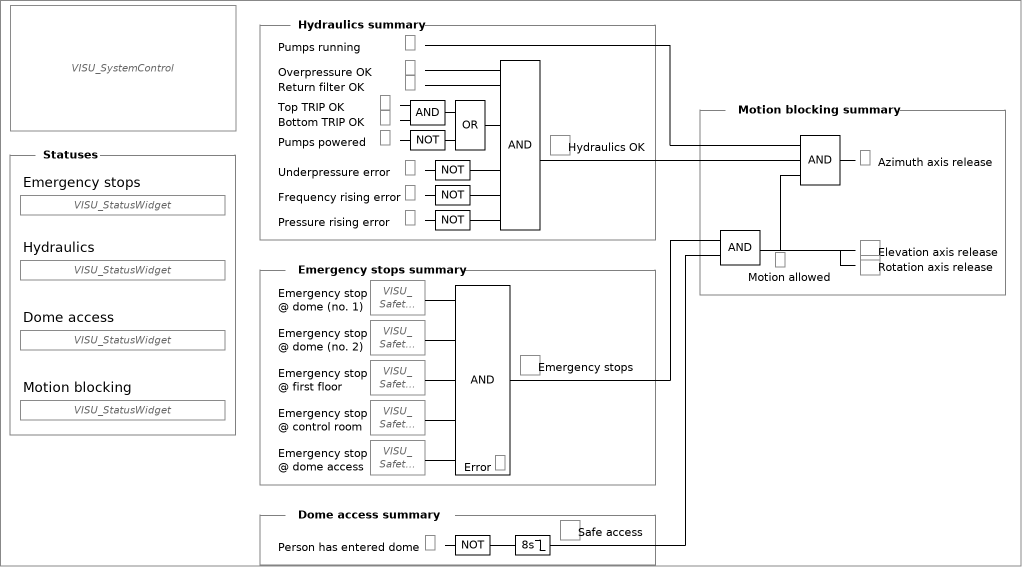
VISUALIZATION VISU_SafetyOverview  // 1022x567
VAR_IN_OUT
	ref : Safety;
    widget : SafetyWidget;
END_VAR
    Polyline (900,110) (1005,110) (1005,295) (700,295) (700,110) (725,110)
    Polyline (455,515) (655,515) (655,565) (260,565) (260,515) (285,515)
    Polyline (425,25) (655,25) (655,240) (260,240) (260,25) (290,25)
    Polyline (465,270) (655,270) (655,485) (260,485) (260,270) (285,270)
    Polyline (100,155) (235,155) (235,435) (10,435) (10,155) (35,155)
    Frame (10,5 226x126)
        shows VISU_SystemControl(status := widget.actualStatus, button_initialize := widget.button_initialize, button_operating := widget.button_operating, button_locking := widget.button_locking)
    Frame (860,150 10x15)
        shows VISU_State_red_green(state := ref.parts.motionBlocking.telescopeAzimuthReleaseOK)
    Label (275,40 120x15), "Pumps running"
    Rectangle (800,135 40x50), "AND"
    Label (875,150 145x25), "Azimuth axis release"
    Line (840,160) (855,160), colour toggle: ref.parts.motionBlocking.telescopeAzimuthReleaseOK
    Frame (405,35 10x15)
        shows VISU_State_gray_green(state := ref.parts.hydraulics.pumpsRunning)
    Frame (370,280 55x35)
        shows VISU_SafetyEmergencyStop(contactNC := ref.parts.emergencyStops.dome1NC, contactNO := ref.parts.emergencyStops.dome1NO)
    Frame (370,320 55x35)
        shows VISU_SafetyEmergencyStop(contactNC := ref.parts.emergencyStops.dome2NC, contactNO := ref.parts.emergencyStops.dome2NO)
    Frame (370,360 55x35)
        shows VISU_SafetyEmergencyStop(contactNC := ref.parts.emergencyStops.firstFloorNC, contactNO := ref.parts.emergencyStops.firstFloorNO)
    Rectangle (455,285 55x190), "AND"
    Frame (495,455 10x15)
        shows VISU_State_green_red(state := ref.parts.emergencyStops.discrepancyError)
    Label (455,455 45x25), "Error"
    Label (275,280 100x40), "Emergency stop @ dome (no. 1)"
    Label (275,320 100x40), "Emergency stop @ dome (no. 2)"
    Label (275,360 100x40), "Emergency stop @ first floor"
    Line (510,380) (670,380), colour toggle: ref.parts.emergencyStops.allOK
    Frame (520,355 20x20)
        shows VISU_State_red_green(state := ref.parts.emergencyStops.allOK)
    Label (535,355 100x25), "Emergency stops"
    Line (425,300) (455,300), colour toggle: ref.parts.emergencyStops.dome1NC
    Line (425,340) (455,340), colour toggle: ref.parts.emergencyStops.dome2NC
    Line (425,380) (455,380), colour toggle: ref.parts.emergencyStops.firstFloorNC
    Line (510,160) (800,160), colour toggle: ref.parts.hydraulics.allOK
    Line (670,240) (670,380), colour toggle: ref.parts.emergencyStops.allOK
    Line (670,240) (720,240), colour toggle: ref.parts.emergencyStops.allOK
    Label (295,15 130x20), "Hydraulics summary"
    Frame (20,195 205x20)
        shows VISU_StatusWidget(widget := widget.emergencyStops.actualStatus)
    Frame (20,260 205x20)
        shows VISU_StatusWidget(widget := widget.hydraulics.actualStatus)
    Frame (20,400 205x20)
        shows VISU_StatusWidget(widget := widget.motionBlocking.actualStatus)
    Label (295,260 170x20), "Emergency stops summary"
    Label (735,100 165x20), "Motion blocking summary"
    Label (40,145 65x20), "Statuses"
    Label (20,170 150x25), "Emergency stops"
    Label (20,235 150x25), "Hydraulics"
    Label (20,375 150x25), "Motion blocking"
    Frame (550,135 20x20)
        shows VISU_State_red_green(state := ref.parts.hydraulics.allOK)
    Label (565,135 100x25), "Hydraulics OK"
    Rectangle (500,60 40x170), "AND"
    Label (275,65 135x15), "Overpressure OK"
    Frame (405,60 10x15)
        shows VISU_State_red_green(state := ref.parts.hydraulics.noOverpressure)
    Line (425,70) (500,70), colour toggle: ref.parts.hydraulics.noOverpressure
    Label (275,80 135x15), "Return filter OK"
    Frame (405,75 10x15)
        shows VISU_State_green_red(state := ref.parts.hydraulics.returnFilterOverpressure)
    Line (425,85) (500,85), colour toggle: ref.parts.hydraulics.returnFilterOverpressure
    Line (470,195) (500,195), colour toggle: ref.parts.hydraulics.pumpsFrequencyNotRising
    Line (470,220) (500,220), colour toggle: ref.parts.hydraulics.pressureNotRising
    Label (275,190 140x15), "Frequency rising error"
    Label (275,215 125x15), "Pressure rising error"
    Line (470,170) (500,170), colour toggle: ref.parts.hydraulics.underpressureError
    Label (275,165 140x15), "Underpressure error"
    Rectangle (435,160 35x20), "NOT"
    Rectangle (435,185 35x20), "NOT"
    Rectangle (435,210 35x20), "NOT"
    Frame (405,160 10x15)
        shows VISU_State_gray_red(state := ref.parts.hydraulics.underpressureError)
    Frame (405,185 10x15)
        shows VISU_State_gray_red(state := ref.parts.hydraulics.pumpsFrequencyNotRising)
    Frame (405,210 10x15)
        shows VISU_State_gray_red(state := ref.parts.hydraulics.pressureNotRising)
    Line (425,170) (435,170), colour toggle: ref.parts.hydraulics.underpressureError
    Line (425,195) (435,195), colour toggle: ref.parts.hydraulics.pumpsFrequencyNotRising
    Line (425,220) (435,220), colour toggle: ref.parts.hydraulics.pressureNotRising
    Line (425,45) (670,45), colour toggle: ref.parts.hydraulics.pumpsRunning
    Line (670,145) (670,45), colour toggle: ref.parts.hydraulics.pumpsRunning
    Line (670,145) (800,145), colour toggle: ref.parts.hydraulics.pumpsRunning
    Label (20,305 150x25), "Dome access"
    Frame (20,330 205x20)
        shows VISU_StatusWidget(widget := widget.domeAccess.actualStatus)
    Label (295,505 170x20), "Dome access summary"
    Label (275,535 150x25), "Person has entered dome"
    Label (275,400 100x40), "Emergency stop @ control room"
    Rectangle (720,230 40x35), "AND"
    Frame (370,400 55x35)
        shows VISU_SafetyEmergencyStop(contactNC := ref.parts.emergencyStops.controlRoomNC, contactNO := ref.parts.emergencyStops.controlRoomNO)
    Line (425,420) (455,420), colour toggle: ref.parts.emergencyStops.controlRoomNC
    Frame (370,440 55x35)
        shows VISU_SafetyEmergencyStop(contactNC := ref.parts.emergencyStops.domeAccessNC, contactNO := ref.parts.emergencyStops.domeAccessNO)
    Line (425,460) (455,460), colour toggle: ref.parts.emergencyStops.domeAccessNC
    Label (275,440 100x40), "Emergency stop @ dome access"
    Line (445,545) (455,545), colour toggle: ref.parts.domeAccess.personHasEntered
    Rectangle (455,535 35x20), "NOT"
    Frame (425,535 10x15)
        shows VISU_State_gray_red(state := ref.parts.domeAccess.personHasEntered)
    Label (745,270 120x15), "Motion allowed"
    Frame (775,252 10x15)
        shows VISU_State_red_green(state := ref.parts.motionBlocking.motionAllowed)
    Line (760,250) (855,250), colour toggle: ref.parts.motionBlocking.motionAllowed
    Line (780,175) (780,250), colour toggle: ref.parts.motionBlocking.motionAllowed
    Line (780,175) (800,175), colour toggle: ref.parts.motionBlocking.motionAllowed
    Frame (860,240 20x20)
        shows VISU_State_red_green(state := ref.parts.motionBlocking.telescopeElevationReleaseOK)
    Label (875,240 145x25), "Elevation axis release"
    Frame (860,255 20x20)
        shows VISU_State_red_green(state := ref.parts.motionBlocking.telescopeRotationReleaseOK)
    Label (875,255 145x25), "Rotation axis release"
    Line (840,250) (840,265), colour toggle: ref.parts.motionBlocking.motionAllowed
    Line (840,265) (855,265), colour toggle: ref.parts.motionBlocking.motionAllowed
    Line (490,545) (515,545), colour toggle: ref.parts.domeAccess.personHasEntered
    Label (275,100 135x15), "Top TRIP OK"
    Frame (380,95 10x15)
        shows VISU_State_red_green(state := ref.parts.hydraulics.topTripOK)
    Line (400,105) (410,105), colour toggle: ref.parts.hydraulics.topTripOK
    Label (275,115 135x15), "Bottom TRIP OK"
    Frame (380,110 10x15)
        shows VISU_State_red_green(state := ref.parts.hydraulics.bottomTripOK)
    Line (400,120) (410,120), colour toggle: ref.parts.hydraulics.bottomTripOK
    Rectangle (410,100 35x25), "AND"
    Frame (380,130 10x15)
        shows VISU_State_gray_green(state := ref.parts.hydraulics.pumpsPowered)
    Line (400,140) (410,140), colour toggle: ref.parts.hydraulics.pumpsPowered
    Label (275,135 100x15), "Pumps powered"
    Rectangle (410,130 35x20), "NOT"
    Line (445,140) (460,140), colour toggle: ref.parts.hydraulics.pumpsPowered
    Rectangle (455,100 30x50), "OR"
    Line (485,125) (500,125), colour toggle: ref.parts.hydraulics.pumpsPowered OR (ref.parts.hydraulics.topTripOK AND ref.parts.hydraulics.bottomTripOK)
    Line (445,112) (455,112), colour toggle: ref.parts.hydraulics.topTripOK AND ref.parts.hydraulics.bottomTripOK
    Rectangle (515,535 35x20), "8s"
    Polyline (535,540) (540,540) (540,550) (545,550)
    Line (685,255) (685,545), colour toggle: ref.parts.domeAccess.safeAccess
    Line (550,545) (685,545), colour toggle: ref.parts.domeAccess.safeAccess
    Line (685,255) (720,255), colour toggle: ref.parts.domeAccess.safeAccess
    Frame (560,520 20x20)
        shows VISU_State_red_green(state := ref.parts.domeAccess.safeAccess)
    Label (575,520 80x25), "Safe access"
END_VISUALIZATION

(* stored: Version 1.1.0.1, ProductVersion 3.1.4019.2
   Visu VISU_SafetyOverview: Id {251cd130-11ba-4afe-9566-a9ce18bac9c1} *)
